KUKA KRL program: check_tool_masref.src, check_tool_masref.dat

--- check_tool_masref.src ---
&ACCESS RVO1
&REL 4
&PARAM TEMPLATE = C:\KRC\Roboter\Template\vorgabe
&PARAM EDITMASK = *
DEF CHECK_TOOL_MASREF( )

;FOLD ; STATION P13060;%{PE}%R 8.2.20,%MKUKATPBASIS,%CCOMMENT,%VNORMAL,%P 2:STATION  P13060
;ENDFOLD
;FOLD ; ROBOT 5;%{PE}%R 8.2.20,%MKUKATPBASIS,%CCOMMENT,%VNORMAL,%P 2:ROBOT 5
;ENDFOLD
;FOLD ; MODULO DE CHECAGEM DE FERRAMENTA;%{PE}%R 8.2.20,%MKUKATPBASIS,%CCOMMENT,%VNORMAL,%P 2:MODULO  DE  CHECAGEM  DE  FERRAMENTA
;ENDFOLD

;  !! ROBO DEVE INICIAR CICLO COM FERRAMENTA C1 !!
;  !!   CASO ESTEJA COM A FERRAMENTA CHECK      !!
;  !!      OS SINAIS DE DOCK OCUPADO            !!

WAIT FOR (NOT $IN[161]) AND ($IN[169]) AND ($IN[177]) AND ($IN[185]) AND ($IN[219])

END

--- check_tool_masref.dat ---
&ACCESS RVO1
&REL 4
&PARAM TEMPLATE = C:\KRC\Roboter\Template\vorgabe
&PARAM EDITMASK = *
DEFDAT CHECK_TOOL_MASREF
;FOLD EXTERNAL DECLARATIONS;%{PE}%MKUKATPBASIS,%CEXT,%VCOMMON,%P
;FOLD GRIPPERTECH EXT
  EXT  H50 (INT:IN, INT:IN ,INT:IN ,GRP_TYP:IN)
;ENDFOLD (GRIPPERTECH EXT)
;FOLD SPOTTECH EXT
  EXT  USERSPOT (S_COMMAND  :IN, SPOT_TYPE:IN)
;ENDFOLD (SPOTTECH EXT)
;FOLD BASISTECH EXT;%{PE}%MKUKATPBASIS,%CEXT,%VEXT,%P
EXT  BAS (BAS_COMMAND  :IN,REAL  :IN )
DECL INT SUCCESS
;ENDFOLD (BASISTECH EXT)
;FOLD USER EXT;%{E}%MKUKATPUSER,%CEXT,%VEXT,%P
;Make your modifications here

;ENDFOLD (USER EXT)
;ENDFOLD (EXTERNAL DECLARATIONS)
ENDDAT
